Yaskawa INFORM job: R1_W63-A2(130,-90)(JEDENR)KM-OK.JBI

/JOB
//NAME R1_W63-A2(130,-90)(JEDENR)KM-OK
///FOLDERNAME KRIS-SCIANA
//POS
///NPOS 109,109,0,5,0,0
///TOOL 0
///POSTYPE PULSE
///PULSE
C00000=63639,-75448,-57109,-45781,44405,-52131
C00001=94617,-44761,-17381,-50840,21971,-50320
C00002=94032,-38268,-10140,-52496,20938,-49575
C00003=93501,-34314,-6346,-52601,20454,-49570
C00004=93501,-33696,-5020,-53682,20144,-49056
C00005=93501,-34730,-7247,-51879,20668,-49913
C00006=94060,-31578,-4114,-53096,20785,-49286
C00007=96769,-33900,-736,-77115,20483,-38452
C00008=95613,-42258,-10455,-72271,20201,-40872
C00009=114836,-25735,13136,-94907,47591,-35443
C00010=113994,-25195,14177,-95513,47040,-35198
C00011=113416,-25115,14231,-95692,46650,-35188
C00012=114835,-25299,14106,-95251,47609,-35212
C00013=114836,-25735,13136,-94907,47591,-35443
C00014=120475,-35953,-1370,-90254,51436,-37673
C00015=139903,-55423,-18281,-79986,42519,-40432
C00016=137225,-49893,-12147,-81254,40513,-40051
C00017=135734,-44853,-8428,-81025,39552,-40397
C00018=135734,-43954,-6692,-81758,39441,-39971
C00019=135733,-44118,-7020,-81616,39462,-40054
C00020=135733,-44152,-7085,-81590,39466,-40071
C00021=135487,-42201,-5602,-81504,39314,-40155
C00022=135051,-44549,-7816,-81347,39046,-40303
C00023=137549,-28607,9365,-88397,55747,-44205
C00024=139027,-39027,1145,-88234,56734,-44007
C00025=137476,-39506,859,-88663,55676,-44006
C00026=139027,-39027,1145,-88234,56734,-44007
C00027=137549,-29554,7549,-87969,55789,-44554
C00028=148111,-23444,13104,-85705,62970,-44063
C00029=149452,-24752,11123,-85135,63945,-44289
C00030=152843,-27774,6403,-83810,66439,-44814
C00031=190226,-72414,-43906,-76175,93946,-45874
C00032=161209,-108399,-80251,-28334,56751,1893
C00033=144499,-103217,-75669,-1877,44915,17731
C00034=128729,-75448,-61988,39008,44461,40651
C00035=127704,-59864,-42449,54687,37585,47688
C00036=129098,-54028,-36168,54912,36254,47616
C00037=129628,-51692,-33607,55058,35721,47558
C00038=128853,-41055,-35233,41549,49027,56551
C00039=128853,-40816,-34294,41807,48684,56370
C00040=128840,-40622,-34262,41768,48749,56399
C00041=128741,-38931,-33203,41693,48960,56453
C00042=128840,-40834,-35088,41540,49052,56556
C00043=127247,-51490,-28798,68208,35092,41834
C00044=107460,-35727,-14488,83818,61987,41705
C00045=109481,-36824,-10898,85519,60200,40359
C00046=110081,-36960,-10983,85600,59771,40373
C00047=108896,-36684,-10810,85439,60617,40344
C00048=109015,-34543,-15794,83164,61082,42520
C00049=120041,-69321,-43674,69014,34434,47015
C00050=122136,-63308,-37796,69130,32837,47090
C00051=122861,-57682,-33939,68142,32556,47661
C00052=122861,-56927,-32189,69156,32288,47121
C00053=122861,-57007,-32371,69051,32315,47177
C00054=122813,-54434,-30992,68368,32532,47537
C00055=123554,-57398,-33775,67835,32116,47869
C00056=119901,-43791,-19123,84492,47521,48262
C00057=120598,-53565,-25534,85539,46900,47634
C00058=121289,-53563,-25533,85597,46409,47669
C00059=119821,-53557,-25530,85473,47449,47596
C00060=108619,-40866,-16292,83893,55508,47491
C00061=107291,-42314,-18146,83526,56507,47634
C00062=103890,-45742,-22613,82683,59075,47961
C00063=65358,-57443,-36501,72798,55432,58639
C00064=52417,-22993,-11744,62287,40232,70223
C00065=52448,-21520,-7613,64192,39368,69108
C00066=53524,-20826,-9330,62266,39348,70274
C00067=54268,-9828,-4864,53802,46811,75130
C00068=54705,-17968,-5209,63027,38079,69889
C00069=54982,-17870,-5950,62349,38146,70289
C00070=79534,-47396,-31619,40921,33509,83414
C00071=77055,-57327,-41840,41672,35586,82928
C00072=52399,-21595,-7667,64214,39397,69093
C00073=52280,-10203,19177,86543,30990,50668
C00074=65588,-27012,-3338,53743,24830,65341
C00075=53020,-9869,18363,85474,30545,51311
C00076=52731,-9659,19405,86358,30690,50818
C00077=54113,-4524,13220,58282,32426,62063
C00078=50068,4464,23038,66171,33858,58581
C00079=51235,8319,32541,84024,22043,48203
C00080=47301,-19438,5291,81944,23802,49722
C00081=53563,-8197,20744,101221,17253,42714
C00082=52099,-17044,3865,82598,33249,58634
C00083=52491,-21454,-7566,64173,39342,69122
C00084=58082,-75430,-54583,50896,47163,49014
C00085=107090,-97721,-77006,13083,48945,24888
C00086=176270,-89310,-67424,-43563,50998,-31527
C00087=192397,-7473,12373,-70971,39141,-64616
C00088=198057,8223,22470,-69865,43596,-64795
C00089=193709,19970,27704,-53252,44315,-71177
C00090=189908,-4171,13998,-69688,37731,-65566
C00091=190186,-4090,14904,-70371,37727,-65154
C00092=177333,-20602,-5731,-45351,35237,-76680
C00093=175050,-24243,-8327,-44090,33896,-77488
C00094=192590,-382,17323,-71128,53739,-66386
C00095=192440,-7538,12322,-71539,53432,-66088
C00096=192407,-7488,12361,-70973,39147,-64614
C00097=174974,-21926,-5725,-35123,23772,-80242
C00098=188989,-2051,16572,-69929,27423,-64375
C00099=188718,-2123,15673,-68886,27437,-64920
C00100=187793,4703,16407,-48977,27446,-71265
C00101=189098,15899,35453,-81248,14956,-53772
C00102=185796,4065,21904,-69855,10987,-63072
C00103=187637,506,18883,-71759,12230,-62079
C00104=192876,-31132,-18558,-63430,41295,-68875
C00105=194286,-74397,-52359,-65330,41559,-67675
C00106=215389,-105846,-76547,-70055,55098,-63190
C00107=223584,-169575,-131522,-59382,5921,-72840
C00108=-821,-169575,-131522,-59382,5921,-72840
BC00000=136785,1186282,980153
BC00001=139225,1191142,956660
BC00002=139225,1191142,956660
BC00003=139225,1191142,956660
BC00004=139225,1191142,956660
BC00005=139225,1191142,956660
BC00006=139225,1191142,956660
BC00007=139225,1191142,956660
BC00008=139225,1191142,956660
BC00009=139225,1191142,956660
BC00010=139225,1191142,956660
BC00011=139225,1191142,956660
BC00012=139225,1191142,956660
BC00013=139225,1191142,956660
BC00014=139225,1191142,956660
BC00015=330193,1191142,950638
BC00016=330193,1191142,950638
BC00017=330193,1191142,950638
BC00018=330193,1191142,950638
BC00019=330193,1191142,950638
BC00020=330193,1191142,950638
BC00021=330193,1191142,950638
BC00022=330193,1191142,950638
BC00023=330193,1191142,950638
BC00024=330193,1191142,950638
BC00025=330193,1191142,950638
BC00026=330193,1191142,950638
BC00027=330193,1191142,950638
BC00028=330193,1191142,950638
BC00029=330193,1191142,950638
BC00030=330193,1191142,950638
BC00031=330193,1191142,950638
BC00032=299174,1191142,906181
BC00033=286767,1191142,888398
BC00034=268383,1191142,862048
BC00035=262048,1191142,852969
BC00036=262048,1191142,852969
BC00037=262048,1191142,852969
BC00038=262048,1191142,852969
BC00039=262048,1191142,852969
BC00040=262048,1191142,852969
BC00041=262048,1191142,852969
BC00042=262048,1191142,852969
BC00043=262048,1191142,852969
BC00044=262048,1191142,852969
BC00045=262048,1191142,852969
BC00046=262048,1191142,852969
BC00047=262048,1191142,852969
BC00048=262048,1191142,852969
BC00049=135922,1191142,844721
BC00050=135922,1191142,844721
BC00051=135922,1191142,844721
BC00052=135922,1191142,844721
BC00053=135922,1191142,844721
BC00054=135922,1191142,844721
BC00055=135922,1191142,844721
BC00056=135922,1191142,844721
BC00057=135922,1191142,844721
BC00058=135922,1191142,844721
BC00059=135922,1191142,844721
BC00060=135922,1191142,844721
BC00061=135922,1191142,844721
BC00062=135922,1191142,844721
BC00063=136156,1191142,864372
BC00064=136347,1191142,880373
BC00065=169794,1191142,879447
BC00066=169434,1191142,871584
BC00067=169145,1191142,865268
BC00068=168763,1191142,856941
BC00069=168763,1191142,856941
BC00070=169058,1191142,863371
BC00071=169058,1191142,863371
BC00072=131278,1191142,880604
BC00073=183941,1191142,964264
BC00074=184826,1186241,942396
BC00075=184854,1186087,941709
BC00076=184854,1186087,941709
BC00077=184853,1186094,941739
BC00078=184853,1186089,941719
BC00079=184853,1186088,941711
BC00080=188555,1183807,935623
BC00081=192324,1185601,940259
BC00082=200209,1189603,895613
BC00083=203241,1191142,878441
BC00084=183401,1191142,887418
BC00085=216255,1191142,901172
BC00086=278220,1191142,927112
BC00087=311263,1191142,940945
BC00088=311915,1191142,924835
BC00089=312176,1191142,918390
BC00090=312176,1191142,918390
BC00091=312176,1191142,918390
BC00092=312176,1191142,918390
BC00093=312176,1191142,918390
BC00094=319915,1191142,925887
BC00095=317231,1191142,941136
BC00096=277815,1191142,941719
BC00097=267276,1191140,907491
BC00098=269255,1191142,910021
BC00099=269255,1191142,910021
BC00100=267276,1191140,907491
BC00101=267276,1191140,907491
BC00102=258620,1191142,890321
BC00103=261384,1191142,905431
BC00104=270057,1191142,869372
BC00105=270057,1191142,869372
BC00106=270057,1191142,869372
BC00107=270057,1191142,1065762
BC00108=218839,1299400,1065762
///POSTYPE BASE
///RECTAN
///RCONF 0,0,0,0,0,0,0,0,0,0,0,0,0,0,0,0,0,0,0,0,0,0,0,0
P00006=0.222,-3.123,-1.508,0.0000,0.0000,0.0000
P00021=-0.225,-6.128,-0.405,0.0000,0.0000,0.0000
P00022=0.222,-3.123,-1.508,0.0000,0.0000,0.0000
P00023=0.143,-0.036,0.682,0.0000,0.0000,0.0000
P00024=0.145,-0.552,1.326,0.0000,0.0000,0.0000
//INST
///DATE 2024/07/25 16:39
///ATTR SC,RW
///GROUP1 RB1,BS1
NOP
'r1_W63-A2(130,-90)(JEDENROBOT)
'Path S1365
SFTOF
MOVJ C00000 BC00000 VJ=20.00
MOVJ C00001 BC00001 VJ=20.00
MOVJ C00002 BC00002 VJ=20.00
MOVL C00003 BC00003 V=60.0
REFP 3 C00004 BC00004
CALL JOB:SEARCH-R1
SET P023 P006
SFTON P023
MOVL C00005 BC00005 V=60.0
REFP 3 C00006 BC00006
CALL JOB:SEARCH-R1
SET P023 P006
SFTON P023
MOVL C00007 BC00007 V=60.0
MOVL C00008 BC00008 V=60.0
MOVL C00009 BC00009 V=100.0
MOVL C00010 BC00010 V=60.0
REFP 3 C00011 BC00011
CALL JOB:SEARCH-R1
SET P023 P006
SFTON P023
MOVL C00012 BC00012 V=60.0
MOVL C00013 BC00013 V=100.0
MOVL C00014 BC00014 V=166.7
'Path S1366
SFTOF
MOVJ C00015 BC00015 VJ=20.00
MOVJ C00016 BC00016 VJ=20.00
MOVL C00017 BC00017 V=60.0
REFP 3 C00018 BC00018
CALL JOB:SEARCH-R1
SET P024 P006
SFTON P024
MOVL C00019 BC00019 V=60.0
MOVL C00020 BC00020 V=60.0
REFP 3 C00021 BC00021
CALL JOB:SEARCH-R1
SET P024 P006
SFTON P024
MOVL C00022 BC00022 V=60.0
MOVL C00023 BC00023 V=100.0
MOVL C00024 BC00024 V=60.0
REFP 3 C00025 BC00025
CALL JOB:SEARCH-R1
SET P024 P006
SFTON P024
MOVL C00026 BC00026 V=60.0
MOVL C00027 BC00027 V=100.0
MOVL C00028 BC00028 V=100.0
MOVL C00029 BC00029 V=100.0
MOVL C00030 BC00030 V=166.7
'Path VIA1504
SFTOF
MOVJ C00031 BC00031 VJ=20.00
'Path VIA1509
SFTOF
MOVJ C00032 BC00032 VJ=20.00
'Path VIA1505
SFTOF
MOVJ C00033 BC00033 VJ=20.00
'Path S1414
SFTOF
MOVJ C00034 BC00034 VJ=20.00
MOVJ C00035 BC00035 VJ=20.00
MOVJ C00036 BC00036 VJ=20.00
MOVL C00037 BC00037 V=100.0
MOVL C00038 BC00038 V=60.0
REFP 3 C00039 BC00039
CALL JOB:SEARCH-R1
SET P021 P006
SFTON P021
MOVL C00040 BC00040 V=60.0
REFP 3 C00041 BC00041
CALL JOB:SEARCH-R1
SET P021 P006
SFTON P021
MOVL C00042 BC00042 V=60.0
MOVL C00043 BC00043 V=100.0
MOVL C00044 BC00044 V=100.0
MOVL C00045 BC00045 V=60.0
REFP 3 C00046 BC00046
CALL JOB:SEARCH-R1
SET P021 P006
SFTON P021
MOVL C00047 BC00047 V=60.0
MOVL C00048 BC00048 V=100.0
'Path S1416
SFTOF
MOVJ C00049 BC00049 VJ=20.00
MOVJ C00050 BC00050 VJ=20.00
MOVL C00051 BC00051 V=60.0
REFP 3 C00052 BC00052
CALL JOB:SEARCH-R1
SET P022 P006
SFTON P022
MOVL C00053 BC00053 V=60.0
REFP 3 C00054 BC00054
CALL JOB:SEARCH-R1
SET P022 P006
SFTON P022
MOVL C00055 BC00055 V=60.0
MOVL C00056 BC00056 V=100.0
MOVL C00057 BC00057 V=60.0
REFP 3 C00058 BC00058
CALL JOB:SEARCH-R1
SET P022 P006
SFTON P022
MOVL C00059 BC00059 V=60.0
MOVL C00060 BC00060 V=100.0
MOVL C00061 BC00061 V=100.0
MOVL C00062 BC00062 V=166.7
'Path VIA1506
SFTOF
MOVJ C00063 BC00063 VJ=20.00
'Path W1380
SFTOF
SFTON P023
MOVJ C00064 BC00064 VJ=20.00
SFTOF
SFTON P023
MOVJ C00065 BC00065 VJ=20.00
MOVJ C00066 BC00066 VJ=20.00
MOVL C00067 BC00067 V=100.0 PL=0
REFP 1 C00068 BC00068
REFP 2 C00069 BC00069
MACRO1 MJ#(0) ARGF9
ARCON
MOVL C00070 BC00070 V=10.0
ARCOF
MOVL C00071 BC00071 V=100.0
MOVL C00072 BC00072 V=166.7
SFTOF
'Path W1378
SFTOF
SFTOF
SFTON P024
MOVJ C00073 BC00073 VJ=20.00
MOVL C00074 BC00074 V=100.0 PL=0
REFP 1 C00075 BC00075
REFP 2 C00076 BC00076
MACRO1 MJ#(0) ARGF9
ARCON
MOVL C00077 BC00077 V=10.0
MOVL C00078 BC00078 V=10.0
MOVL C00079 BC00079 V=10.5
ARCOF
MOVL C00080 BC00080 V=100.0
MOVL C00081 BC00081 V=166.7
SFTOF
'Path VIA1510
SFTOF
MOVJ C00082 BC00082 VJ=20.00
'Path W1379
SFTOF
SFTON P024
MOVJ C00083 BC00083 VJ=20.00
SFTOF
'Path VIA1507
SFTOF
MOVJ C00084 BC00084 VJ=20.00
'Path VIA1508
SFTOF
MOVJ C00085 BC00085 VJ=20.00
MOVJ C00086 BC00086 VJ=20.00
'Path W1432
SFTOF
SFTON P021
MOVJ C00087 BC00087 VJ=20.00
MOVJ C00088 BC00088 VJ=20.00
MOVL C00089 BC00089 V=100.0 PL=0
REFP 1 C00090 BC00090
REFP 2 C00091 BC00091
MACRO1 MJ#(0) ARGF9
ARCON
MOVL C00092 BC00092 V=9.2
MOVL C00093 BC00093 V=9.2
ARCOF
MOVL C00094 BC00094 V=100.0
MOVL C00095 BC00095 V=166.7
SFTOF
'Path W1433
SFTOF
SFTON P021
MOVJ C00096 BC00096 VJ=20.00
SFTOF
'Path W1434
SFTOF
SFTON P021
MOVL C00097 BC00097 V=100.0 PL=0
REFP 1 C00098 BC00098
REFP 2 C00099 BC00099
MACRO1 MJ#(0) ARGF9
ARCON
SFTON P022
MOVL C00100 BC00100 V=9.2
MOVL C00101 BC00101 V=9.2
ARCOF
MOVL C00102 BC00102 V=100.0
MOVL C00103 BC00103 V=166.7
SFTOF
'Path W1435
MOVL C00104 BC00104 V=100.0
MOVL C00105 BC00105 V=166.7
SFTOF
MOVJ C00106 BC00106 VJ=20.00
MOVJ C00107 BC00107 VJ=100.00
MOVJ C00108 BC00108 VJ=100.00
END
